TYPE ST_CommandConfiguration :
STRUCT
	CommandConfiguration : REFERENCE	TO ST_CommandConfiguration;
	ComponentName          : STRING;
	ComponentTyoe          : STRING;
	CommandCount           : DINT;
	
END_STRUCT
END_TYPE

(* stored: Version 1.1.0.1
   DUT ST_CommandConfiguration: Id {616dc179-725c-4eb3-8095-d170339ad288} *)
